PROGRAM Kytkin
VAR
	RS_0: RS; //kytkin pitäis laittaa punanen valo päälle ekalla painannalla, ja sitten sammuttaaa se seuraavalla painalluksella. Mutta nyt se jää vain päälle.
	TON_0: TON;
	L: INT;
	NAPITUS: CTU;
END_VAR

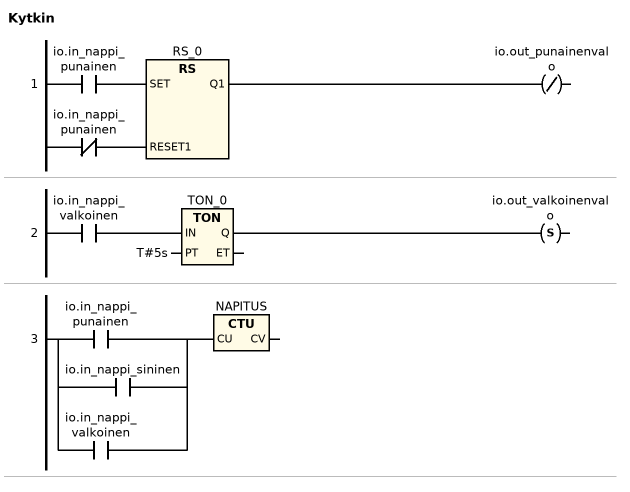
// NETWORK 1
RS_0(SET := io.in_nappi_punainen, RESET1 := NOT io.in_nappi_punainen); // RS
io.out_punainenvalo := NOT RS_0.Q1;

// NETWORK 2
TON_0(IN := io.in_nappi_valkoinen, PT := T#5s); // TON
io.out_valkoinenvalo S= TON_0.Q;

// NETWORK 3
NAPITUS(CU := io.in_nappi_punainen OR io.in_nappi_sininen OR io.in_nappi_valkoinen); // CTU

END_PROGRAM

(* stored: Version 1.1.0.1, ProductVersion 3.1.4024.10
   POU Kytkin: Id {e3635ed3-b249-48d8-b741-451a8aa85b97}, SpecialFunc None *)
